// TwinCAT 3 PLC project Main
// ProgramVersion: 3.1.4024.12
// libraries:
//   Tc2_Standard, * (Beckhoff Automation GmbH)
//   Tc2_System, * (Beckhoff Automation GmbH)
//   Tc3_Module, * (Beckhoff Automation GmbH)
// project tree:
//   DUTs/ GEMMA.TcDUT
//   / GlobalTextList.TcGTLO, PlcTask.TcTTO, Visualization Manager.TcVMO (not stored)
//   POUs/ FB_Clock.TcPOU, FB_Coordinador_ST.TcPOU, FB_Coordinador_SFC.TcPOU, FB_Director_ST.TcPOU, FB_Discharger_SFC.TcPOU, FB_Discharger_ST.TcPOU, FB_Object_Template_SFC.TcPOU, FB_Object_Template_ST.TcPOU, FB_Panel.TcPOU, MAIN.TcPOU
//   VISUs/ Visualization.TcVIS

CONFIGURATION Main
    RESOURCE PLC ON TwinCAT3
        TASK PlcTask(INTERVAL := T#10ms, PRIORITY := 20);
        PROGRAM MAIN WITH PlcTask : MAIN;
    END_RESOURCE
END_CONFIGURATION

// ---- DUTs/GEMMA.TcDUT

TYPE GEMMA :
(
	  (* Modes de la Guia de Estudio de los Modes de Marcha y Parada *)
    (* [Modes du Guide d'Etude des Modes de Marche et d'Arrêt] *)
    (* [Modes of Study Guide of the Modes of Operating and Stopping] *)

    (* Procedimientos de parada [les procédures d'arrets/stop procedures] *)
    A1ParadaInicial, (*  0: parada en el estado inicial
               [arrêt dans etat initial] 
               [stopped in the initial state] *)
    A2ParaFinCiclo, (*  1: parada solicitada a final de ciclo
               [arret demandé en fin de cycle] 
               [requested end cycle stop] *)
    A3ParadaEstado, (*  2: parada solicitada en un estado determinado
               [arret demande dans etat determine] 
               [requested particular state stop] *)
    A4ParadaObtenida, (*  3: parada obtenida
               [arret obtenu] 
               [obteined stop] *)
    A5PreparandoTrasFallo, (*  4: preparacion para la recuperacion del fallo
               [preparation pour remise en route apres defaillance] 
               [preparation for the recovery of the Fail] *)
    A6Inicializando, (*  5: situando la PO en el estado inicial
               [mise PO dans état initial] 
               [set the PO in initial state] *)
    A7SituandoEstado, (*  6: situando la PO en un estado determinado
               [mise PO dans état déterminé]
               [set the PO in a certain state] *)

    (* Procedimientos de funcionamiento [les procédures de fonctionnement/operating procedures] *)
    F1ProduccionNormal, (*  7: produccion normal
               [production normale] 
               [normal operation] *)
    F2SecuenciaPreparacion, (*  8: secuencia de preparacion
               [marche de preparation] 
               [preparation sequence] *)
    F3SecuenciaFinalizacion, (*  9: secuencia de finalizacion
               [marche de cloture] 
               [ending sequence] *)
    F4VerificacionSinOrden, (* 10: verificacion en desorden
               [marche de verification dans le desordre] 
               [verification with no order] *)
    F5VerificacionOrdenada, (* 11: verificacion en orden
               [marche de verification dans l'ordre] 
               [verification whit order] *)
    F6Probando, (* 12: prueba
               [marche de test] 
               [test] *)

    (* Procedimientos de fallo [les procédures en défaillances] *)
    D1ParadaEmergencia, (* 13: parada de emergencia
               [arret d'urgence] 
               [emergency stop] *)
    D2TratamientoFallos, (* 14: diagnostico y/o tratamiento de los fallos
               [diagnostic et/ou traitement de la défaillance] 
               [diagnosis and/or treatment of Fails] *)
    D3ProducirConFallos  (* 15: produccion a pesar de los fallos
               [production tout de même] 
               [production despite the Fails] *)
);
END_TYPE

// ---- POUs/MAIN.TcPOU
PROGRAM MAIN
VAR
END_VAR

END_PROGRAM

// ---- POUs/FB_Clock.TcPOU
FUNCTION_BLOCK FB_Clock
(*
Copyright (c) 2009-2017 victortorreslopez
GNU General Public License
*)
VAR_INPUT
  EN: BOOL := TRUE;	(* ENabled *)
  PT: TIME := T#500ms; (* Semicycle time *)
END_VAR
VAR_OUTPUT
  ET: TIME; (* Elapsed time *)
  Q: BOOL; (* Square wave *)
END_VAR
VAR
  Timer: TON; (* Auto-pilot timer *)
END_VAR

(* OUTPUT FUNCTION *)
IF Timer.Q THEN
  Q := NOT Q;
END_IF

(* FUNCTION BLOCKS *)
Timer(IN := EN AND NOT Timer.Q, PT := PT, ET => ET);

END_FUNCTION_BLOCK

// ---- POUs/FB_Coordinador_ST.TcPOU
FUNCTION_BLOCK FB_Coordinador_ST
VAR_INPUT
	Tray_1 : BOOL; 
	Tray_2 : BOOL;
END_VAR
VAR_OUTPUT
	IC : BOOL;
	Fail : BOOL;
	Pause : BOOL;
	Mode := GEMMA;
END_VAR

END_VAR
VAR
	Director : FB_Director_ST;
	Coordinador : FB_Coordinador_SFC;
	Discharger : FB_Discharger_ST;
	ModeAns : GEMMA;
	Panel : FB_Panel;
	
END_VAR

Director(IC:= Coordinador.IC, Manual:= Panel.Manual, Go:= Panel.Go, Stop := Panel.Stop,
		 Resume := Panel.Go, Cancel := Panel.Stop, EndBatch := Coordinador.Done,
		 End := Coordinador.End, Fail := Fail);

Panel(Mode := Director.Mode);
		 
Coordinador(Execute:= Director.IC:=Discharger.IC,
			Discharger_Ready:= Discharger.Ready,
			Discharger_Done:= Discharger.Done,
			Tray_1 := Tray_1,
			Tray_2:= Tray_2);
			
// Associate module variables
Discharger (Execute :=Coordinador.Discharger_Execute,
			Ack := NOT (Coordinador.Discharger_Execute),
			Reset := Director.Reset,
			Pause := Director.Pause,
			B1 := Tray_1,
			B2 := Tray_2);

END_FUNCTION_BLOCK

// ---- POUs/FB_Director_ST.TcPOU
FUNCTION_BLOCK FB_Director_ST
VAR_INPUT
	IC: BOOL := TRUE;
	Manual: BOOL;
	Go: BOOL;
	Stop: BOOL;
	Resume: BOOL;
	Cancel: BOOL;
	EndBatch: BOOL;
	//Emergency: BOOL;
	End: BOOL;
	Fail: BOOL;
END_VAR
VAR_OUTPUT
	Mode: GEMMA := GEMMA.A6Inicializando;
	Arret: BOOL;
	Defail: BOOL;
	Fonctionnement: BOOL;
	Pause: BOOL;
	Stopped: BOOL;
	Production: BOOL;
	
END_VAR
VAR
	ModeAns: GEMMA;
END_VAR

Arret := (Mode >= GEMMA.A1ParadaInicial) AND (Mode <= GEMMA.A7SituandoEstado);
Defail := (Mode >= GEMMA.D1ParadaEmergencia) AND (Mode <= GEMMA.D3ProducirConFallos);
Fonctionnement := (Mode >= GEMMA.F1ProduccionNormal) AND (Mode <= GEMMA.F6Probando);
Pause := (Mode = GEMMA.A3ParadaEstado) OR (Mode = GEMMA.A4ParadaObtenida) 
		  OR (Mode = GEMMA.A5PreparandoTrasFallo)OR (Mode = GEMMA.D1ParadaEmergencia)
		  OR (Mode = GEMMA.D2TratamientoFallos);
Stopped := (Mode >= GEMMA.A1ParadaInicial) AND (Mode <= GEMMA.A7SituandoEstado);
Production := (Mode = GEMMA.A2ParaFinCiclo) 
			   OR (Mode = GEMMA.A3ParadaEstado)
			   OR (Mode = GEMMA.F1ProduccionNormal)
			   OR (Mode = GEMMA.F2SecuenciaPreparacion) 
			   OR (Mode = GEMMA.F3SecuenciaFinalizacion) 
			   OR (Mode = GEMMA.F5VerificacionOrdenada)
			   OR (Mode = GEMMA.F6Probando)
			   OR (Mode = GEMMA.D3ProducirConFallos);

CASE Mode OF

	(*GEMMA.A6Inicializando: (* A6 -> A1 o F4 *)
		ModeAns := GEMMA.A6Inicializando;
		IF IC THEN 
			Mode := GEMMA.A1ParadaInicial;
		ELSIF Manual THEN 				
			Mode := GEMMA.F4VerificacionSinOrden;
		END_IF*)

	GEMMA.A1ParadaInicial: (* A1 -> A6, F4, F5, F2 o F6 *)
		ModeAns := GEMMA.A1ParadaInicial;
		IF NOT IC THEN // IF NOT Restaurada THEN
			Mode := GEMMA.A6Inicializando;				
		ELSIF Manual THEN 				
			Mode := GEMMA.F4VerificacionSinOrden;			            
		ELSIF Go THEN
			Mode := GEMMA.F2SecuenciaPreparacion;
		ELSE
			; // Esperar a que se pulse el bortón de marcha
		END_IF
		
	GEMMA.A3ParadaEstado: 
		IF Fail THEN																// A3 -> D2
			Mode := GEMMA.D2TratamientoFallos;
		ELSIF Stop THEN															// A3 -> A4
			Mode := GEMMA.A4ParadaObtenida;
		ELSE
			; // Seguir produciendo hasta que todos los módulos paren en un estado estable
		END_IF
					
	GEMMA.A4ParadaObtenida:	;													// A4 -> retorna
	GEMMA.A5PreparandoTrasFallo:
		IF Resume THEN
			Mode := ModeAns;
		ELSIF Cancel THEN
			Mode := GEMMA.A6Inicializando;
		END_IF; 		
				
	GEMMA.F1ProduccionNormal:	        
		// cambios de modo actual
		IF Fail THEN 															// cualquiera -> D2
			ModeAns := GEMMA.A2ParaFinCiclo;
			Mode := GEMMA.D2TratamientoFallos;
		ELSIF Manual THEN				
			Mode := GEMMA.A3ParadaEstado; 								// cualquiera -> A3
		ELSIF Manual THEN 				
			Mode := GEMMA.F4VerificacionSinOrden;						// cualquiera -> F4
		ELSIF EndBatch THEN 			
			Mode:= GEMMA.F3SecuenciaFinalizacion;
		ELSE                
			; // continuar con la preparación/producción/finalización
		END_IF
		
	GEMMA.F3SecuenciaFinalizacion:
		IF End THEN
			Mode := GEMMA.A1ParadaInicial;
		ELSE 
			;
		END_IF
					
	GEMMA.F4VerificacionSinOrden: (* F4 -> ModePrev *)
		IF Fail THEN
		Mode := GEMMA.D2TratamientoFallos;				
		ELSIF NOT Manual THEN				
			Mode := GEMMA.A6Inicializando; // al salir del modo planta volver al modo previo				
		ELSE                
			; // Seguir en modo manual
		END_IF
	(*GEMMA.D1ParadaEmergencia: (* Parada de emergencia *)
		IF NOT Emergency THEN //  TODO CONSIGNA DE EMERGENCIA DEBE TENER ENCUENTA LA POC
			Mode := GEMMA.A6Inicializando; // Al quitar la parada de emergencia hay que reinicializar la estación
		ELSIF Manual then							// desde A1 se puede entrar F4 para arreglar el problema
			ModeAns := GEMMA.D1ParadaEmergencia;
			Mode := GEMMA.F4VerificacionSinOrden;
		ELSE                
			; // Esperar a que se quite la parada de emergencia
		END_IF*)
		
	GEMMA.D2TratamientoFallos: (* Diagnostico/tratamiento de los fallos *)
		IF NOT Fail THEN // el fallo se resuelve por sí solo (no debería pasar)
			Mode := GEMMA.A5PreparandoTrasFallo;
		ELSIF Manual THEN // se pasa a modo F4 para arreglarlo
			Mode := GEMMA.F4VerificacionSinOrden;
		ELSIF Go THEN // se pulsa Marcha para intentar recuperar                
			Mode := GEMMA.A5PreparandoTrasFallo;
		END_IF


END_CASE

END_FUNCTION_BLOCK

// ---- POUs/FB_Coordinador_SFC.TcPOU
FUNCTION_BLOCK FB_Coordinador_SFC EXTENDS FB_Object_Template_SFC;
VAR_INPUT
// Functions
Produce : BOOL;
//Discharger
	Discharger_Ready: BOOL;
	Discharger_Done: BOOL;
	Tray_1: BOOL;
	Tray_2: BOOL;
END_VAR
VAR_OUTPUT
	//Discharger
	Discharger_Execute: BOOL;
	Discharger_Ack: BOOL;
	

END_VAR
VAR
END_VAR

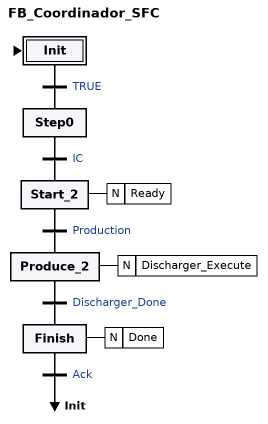
INITIAL_STEP Init:
END_STEP
TRANSITION FROM Init TO Step0
    := TRUE;
END_TRANSITION
STEP Step0:
END_STEP
TRANSITION FROM Step0 TO Start_2
    := IC;
END_TRANSITION
STEP Start_2:
    Ready(N);
END_STEP
TRANSITION FROM Start_2 TO Produce_2
    := Production;
END_TRANSITION
STEP Produce_2:
    Discharger_Execute(N);
END_STEP
TRANSITION FROM Produce_2 TO Finish
    := Discharger_Done;
END_TRANSITION
STEP Finish:
    Done(N);
END_STEP
TRANSITION FROM Finish TO Init
    := Ack;
END_TRANSITION

TRANSITION Production:
Produce AND Execute;
END_TRANSITION

END_FUNCTION_BLOCK

// ---- POUs/FB_Object_Template_SFC.TcPOU
FUNCTION_BLOCK FB_Object_Template_SFC
VAR_INPUT
	// Control variables
	Execute: BOOL;
	Ack: BOOL;
	SFCReset: BOOL; 
	SFCPause: BOOL;
	IC: BOOL;
	// Physical variables
END_VAR
VAR_OUTPUT
	//Control variables
	Ready: BOOL;
	Done: BOOL;
	//Physical Variables
END_VAR
VAR
END_VAR

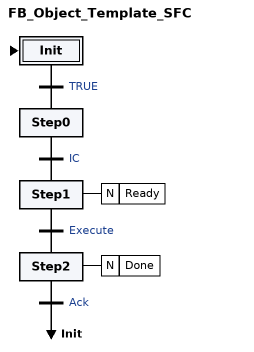
INITIAL_STEP Init:
END_STEP
TRANSITION FROM Init TO Step0
    := TRUE;
END_TRANSITION
STEP Step0:
END_STEP
TRANSITION FROM Step0 TO Step1
    := IC;
END_TRANSITION
STEP Step1:
    Ready(N);
END_STEP
TRANSITION FROM Step1 TO Step2
    := Execute;
END_TRANSITION
STEP Step2:
    Done(N);
END_STEP
TRANSITION FROM Step2 TO Init
    := Ack;
END_TRANSITION

END_FUNCTION_BLOCK

// ---- POUs/FB_Discharger_ST.TcPOU
FUNCTION_BLOCK FB_Discharger_ST EXTENDS FB_Object_Template_ST
VAR_INPUT
	B1: BOOL; 
	B2: BOOL;
	dcha_1 AT %I*: BOOL;
	dcha_2 AT %I*: BOOL;
	izda_1 AT %I*: BOOL;
	izda_2 AT %I*: BOOL;
	arriba AT %I*: BOOL;
	abajo  AT %I*: BOOL;
	cogido AT %I*: BOOL;
END_VAR
VAR_OUTPUT
	avanza_1 AT %Q*: BOOL;
	avanza_2 AT %Q*: BOOL;
	baja	 AT %Q*: BOOL;
	coge 	 AT %Q*: BOOL;
END_VAR
VAR
	Discharger : FB_Discharger_SFC;
END_VAR

//Define initial conditions
IC := izda_1 AND izda_2 AND arriba AND NOT cogido;
//Declare module
Discharger(Execute:=Execute,
		   Ack:=Ack,
		   SFCReset:=Reset,
		   SFCPause:=Pause,
		   IC:=IC,
		   B1:=B1,
		   B2:=B2,
		   dcha_1:=dcha_1,
		   dcha_2:=dcha_2,
		   izda_1:=izda_1,
		   izda_2:=izda_2,
		   arriba:=arriba,
		   abajo:=abajo,
		   cogido:=cogido
);
		   
//Declare module actuators
Ready := Discharger.Ready;
Done := Discharger.Done;
avanza_1 := Discharger.avanza_1;
avanza_2 := Discharger.avanza_2;
baja := Discharger.baja;
coge := Discharger.coge;

END_FUNCTION_BLOCK

// ---- POUs/FB_Object_Template_ST.TcPOU
FUNCTION_BLOCK FB_Object_Template_ST
VAR_INPUT
	// Control variables
	Execute: BOOL;
	Ack: BOOL;
	Reset: BOOL; 
	Pause: BOOL;
	// Physical variables
	
END_VAR
VAR_OUTPUT
	//Control variables
	Ready: BOOL;
	Done: BOOL;
	//Physical Variables
	
END_VAR
VAR
	// Initial conditions
	IC: BOOL := TRUE;
END_VAR

END_FUNCTION_BLOCK

// ---- POUs/FB_Discharger_SFC.TcPOU
FUNCTION_BLOCK FB_Discharger_SFC EXTENDS FB_Object_Template_SFC
VAR_INPUT
	B1: BOOL;
	B2: BOOL;
	dcha_1: BOOL;
	dcha_2: BOOL;
	izda_1: BOOL;
	izda_2: BOOL;
	arriba: BOOL;
	abajo: BOOL;
	cogido: BOOL;
END_VAR
VAR_OUTPUT
	avanza_1: BOOL;
	avanza_2: BOOL;
	baja: BOOL;
	coge: BOOL;
END_VAR
VAR
END_VAR

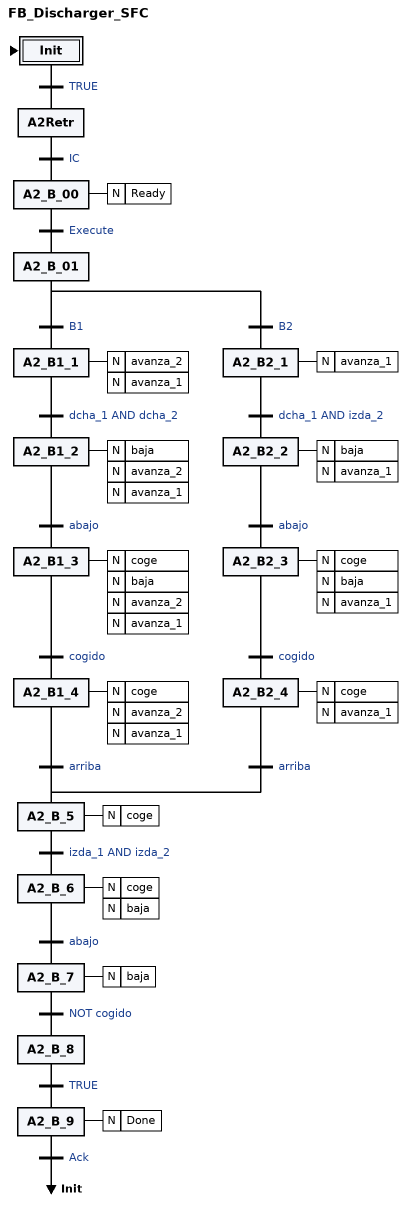
INITIAL_STEP Init:
END_STEP
TRANSITION FROM Init TO A2Retr
    := TRUE;
END_TRANSITION
STEP A2Retr:
END_STEP
TRANSITION FROM A2Retr TO A2_B_00
    := IC;
END_TRANSITION
STEP A2_B_00:
    Ready(N);
END_STEP
TRANSITION FROM A2_B_00 TO A2_B_01
    := Execute;
END_TRANSITION
STEP A2_B_01:
END_STEP
TRANSITION FROM A2_B_01 TO A2_B1_1
    := B1;
END_TRANSITION
STEP A2_B1_1:
    avanza_2(N);
    avanza_1(N);
END_STEP
TRANSITION FROM A2_B1_1 TO A2_B1_2
    := dcha_1 AND dcha_2;
END_TRANSITION
STEP A2_B1_2:
    baja(N);
    avanza_2(N);
    avanza_1(N);
END_STEP
TRANSITION FROM A2_B1_2 TO A2_B1_3
    := abajo;
END_TRANSITION
STEP A2_B1_3:
    coge(N);
    baja(N);
    avanza_2(N);
    avanza_1(N);
END_STEP
TRANSITION FROM A2_B1_3 TO A2_B1_4
    := cogido;
END_TRANSITION
STEP A2_B1_4:
    coge(N);
    avanza_2(N);
    avanza_1(N);
END_STEP
TRANSITION FROM A2_B1_4 TO A2_B_5
    := arriba;
END_TRANSITION
TRANSITION FROM A2_B_01 TO A2_B2_1
    := B2;
END_TRANSITION
STEP A2_B2_1:
    avanza_1(N);
END_STEP
TRANSITION FROM A2_B2_1 TO A2_B2_2
    := dcha_1 AND izda_2;
END_TRANSITION
STEP A2_B2_2:
    baja(N);
    avanza_1(N);
END_STEP
TRANSITION FROM A2_B2_2 TO A2_B2_3
    := abajo;
END_TRANSITION
STEP A2_B2_3:
    coge(N);
    baja(N);
    avanza_1(N);
END_STEP
TRANSITION FROM A2_B2_3 TO A2_B2_4
    := cogido;
END_TRANSITION
STEP A2_B2_4:
    coge(N);
    avanza_1(N);
END_STEP
TRANSITION FROM A2_B2_4 TO A2_B_5
    := arriba;
END_TRANSITION
STEP A2_B_5:
    coge(N);
END_STEP
TRANSITION FROM A2_B_5 TO A2_B_6
    := izda_1 AND izda_2;
END_TRANSITION
STEP A2_B_6:
    coge(N);
    baja(N);
END_STEP
TRANSITION FROM A2_B_6 TO A2_B_7
    := abajo;
END_TRANSITION
STEP A2_B_7:
    baja(N);
END_STEP
TRANSITION FROM A2_B_7 TO A2_B_8
    := NOT cogido;
END_TRANSITION
STEP A2_B_8:
END_STEP
TRANSITION FROM A2_B_8 TO A2_B_9
    := TRUE;
END_TRANSITION
STEP A2_B_9:
    Done(N);
END_STEP
TRANSITION FROM A2_B_9 TO Init
    := Ack;
END_TRANSITION

END_FUNCTION_BLOCK

// ---- POUs/FB_Panel.TcPOU
FUNCTION_BLOCK FB_Panel
FUNCTION_BLOCK FB_Panel

VAR_INPUT
   Modo: GEMMA;
   Restart_Time: TIME := T#3S;

END_VAR
VAR_OUTPUT
	Emergency: BOOL;
	Go:     BOOL;
	Manual:     BOOL;
    Stop:       BOOL;
    Restart:   BOOL; (* Restablece situacion inicial *)
    Restablece: BOOL; (* Restablece la condicion de fallo *)
    Restaura:   BOOL; (* Restaura condiciones iniciales *)
END_VAR
VAR
    (* Bloques funcionales *)
    CLK: FB_Clock;
    Trig_PGo: R_TRIG;
    TmpReinicio: TON;

    (* Entradas *)
    PEmergency AT %I*: BOOL; (* Pulsador de parada de emergencia [EMERGENCY STOP] *)
    PGo AT %I*: BOOL; (* Pulsador de marcha [START] *)
    PStop AT %I*: BOOL := TRUE; (* Pulsador de parada [STOP] *)
    PManual AT %I*: BOOL; (* Selector de modo AUTO/MAN [AUTO/MAN] *)

    (* Salidas *)
    Red_Lamp    AT %Q*: BOOL; (* Lampara de alarma [ALARM] *)
	Yellow_Lamp AT %Q*: BOOL; (* Lampara de alarma [ALARM] *)
	Green_Lamp  AT %Q*: BOOL; (* Lampara de alarma [ALARM] *)
END_VAR

(* PARAMETROS DE SALIDA *)
Emergencia := PEmergency;
Manual := PManual;
Restart := TmpReinicio.Q;
Restablece := PGo;
Restaura := PGo;
Marcha := Trig_PGo.Q;
Para := PStop;

(* ACCIONES *)
Red_Lamp := (Modo = F3SecuenciaFinalizacion) OR (((Modo = D1ParadaEmergencia) OR (Modo = D2TratamientoFallos) OR (Modo = F2SecuenciaPreparacion)) AND CLK.Q);
Yellow_Lamp := ((Modo = A6Inicializando) OR (Modo = D1ParadaEmergencia) OR (Modo = D2TratamientoFallos)) AND CLK.Q;
Green_Lamp := ((Modo = A2ParaFinCiclo) OR (Modo = F1ProduccionNormal) OR (Modo = F2SecuenciaPreparacion) OR (Modo = F3SecuenciaFinalizacion)) OR ((Modo = A1ParadaInicial) AND CLK.Q);

(* BLOQUES FUNCIONALES *)
CLK();

Trig_PGo(CLK := PGo);

TmpReinicio(
    IN := PGo AND NOT PStop,
	PT := Restart_Time
    );

END_FUNCTION_BLOCK

// ---- VISUs/Visualization.TcVIS
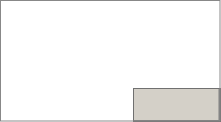
VISUALIZATION Visualization  // 221x122
    Button (133,88 88x34)
END_VISUALIZATION
